Staubli VAL3: Control_PanelD.pgx

public program Control_PanelD()
begin
  call Control_PanelS("",20,0,18,11)


end
